TYPE St_InsulationMonitor_PassThrough :
STRUCT
	b_NetContFB				: BOOL;
	b_MccbfbMaster			: BOOL;
	b_MccbfbSlave			: BOOL;
	b_ACdetected			: BOOL;
	b_PENlinkFB				: BOOL;	
END_STRUCT
END_TYPE

(* stored: Version 1.1.0.1, ProductVersion 3.1.4026.18
   DUT St_InsulationMonitor_PassThrough: Id {5ade6dfc-dcaa-40be-9d98-913c8d8eb56f} *)
